FUNCTION_BLOCK COMM_ADAPTER_PLUG_PROXY_137D8FA9F791DEABB (* Service Interface Function Block Type *)
  (* Standard: 61499-2 *)
  (* Version 0.0, 9/22/2017, bababen, nxtControl GmbH, template *)
  PACKAGE Main;
  (* Compiler Cpp nxtControl builtin 1.0 *)
  {SET_ATTRIBUTE(Configuration.GenericFBType.InterfaceParams, Runtime.System#<InterfaceList> <Plugs> <AdapterDeclaration Name="Out2" Type="BoolAdp" Namespace="Main" /> </Plugs> </InterfaceList>)}
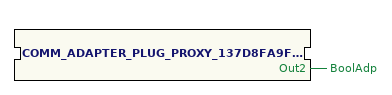
  PLUGS
    Out2 : BoolAdp;
  END_PLUGS
END_FUNCTION_BLOCK
